Staubli VAL3: StaubliSocket.dtx

bool bBool
jointRs jJRs
jointRx jJ
mdesc mNomSpeed
num nPcNum[6]
sio sServer = {link=Socket\clserver}
string sPos
